Staubli VAL3: Main.pjx

--- Main.pjx ---
Parameters version=s7.8.3 stackSize=10000 millimeterUnit=true
Program file=ContorlLight.pgx
Program file=EnterPageKey.pgx
Program file=Init.pgx
Program file=Main.pgx
Program file=MainKey.pgx
Program file=OnF1.pgx
Program file=OnF2.pgx
Program file=OnF3.pgx
Program file=OnF4.pgx
Program file=OnF5.pgx
Program file=OnF6.pgx
Program file=OnF7.pgx
Program file=OnF8.pgx
Program file=Refresh.pgx
Program file=SetPara.pgx
Program file=start.pgx
Program file=stop.pgx
Data file=Main.dtx
Library alias=user path=Disk://userPage/USERPAGE.pjx
Library alias=RobMaster path=Disk://DealRobMaster/DealRobMaster.pjx
Library alias=Prd path=Disk://Product/Product.pjx
Library alias=Pallet path=Disk://Pallet/Pallet.pjx
Library alias=Path path=Disk://Path/Path.pjx
Library alias=Tool path=Disk://Tool/Tool.pjx autoload=false
Library alias=Frame path=Disk://Frame/Frame.pjx autoload=false
Library alias=IO path=Disk://IO/IO.pjx
Library alias=Home path=Disk://Home/Home.pjx autoload=false
Library alias=PublicData path=Disk://PublicData/PublicData.pjx
Library alias=Motion path=Disk://Motion/Motion.pjx
Library alias=SparePoint path=Disk://SparePoint/SparePoint.pjx autoload=false
Library alias=PublicProg path=Disk://PublicProg/PublicProg.pjx
Library alias=prd path=Disk://template/normalPath/normalPath.pjx

--- Main.dtx ---
mdesc mNomSpeed
bool bExit
bool bUserRefresh
aio aAio
string sParameter
string sListItemValue
bool bListRefresh
string sPath

--- Main.pgx ---
program Main()
  local num l_nKey
begin
  //

  do
    call Refresh()
    l_nKey=getKey()
    bUserRefresh=false
    call MainKey(l_nKey)
    delay(0)
  until bExit
end

--- start.pgx ---
program start()
  local num l_nLastId
  local num l_ni
begin
  call Init()
  taskCreate "light",30,ContorlLight()
  wait(taskStatus("light")==1)
  call Main()
end

--- ContorlLight.pgx ---
program ContorlLight()
begin
  //

  while !bExit
    //红灯
    if PublicData:sStatus=="stop"
      IO:dOut["dOut2"]=true
      IO:dOut["dOut3"]=false
      IO:dOut["dOut4"]=false
    elseIf PublicData:sStatus=="pause"
      IO:dOut["dOut2"]=false
      IO:dOut["dOut3"]=false
      IO:dOut["dOut4"]=true
    elseIf PublicData:sStatus=="run"
      IO:dOut["dOut2"]=false
      IO:dOut["dOut3"]=true
      IO:dOut["dOut4"]=false
    endIf
    delay(0)
  endWhile

end

--- EnterPageKey.pgx ---
program EnterPageKey(num& x_nKey, num& x_nSelect, string& x_sItem)
  local string l_sStr
  local num l_nKey
  local string l_sEmpty
  local string l_sValue
  local num l_nItem
  local num l_nView
  local string l_sItem
  local point lp
  local string l_sYN[2]
  local bool l_bRes
  local num l_nTemp
  local num l_i
begin
  //
  //编辑项目
  switch x_nSelect
    //
    case 0

    break
    //砂带补偿量
    default
      if x_nKey==270
        call user:editNum(x_sItem,sListItemValue[x_nSelect],l_nTemp,x_nSelect)
        if l_nTemp>0.08
          popUpMsg("最大0.08")
          l_nTemp=0.08
          sParameter[x_nSelect]=sPath[x_nSelect-1]
          sListItemValue[0]=toString(".4",PublicData:nDelta)
          call user:strlength(sParameter[l_i],user:nBottomX/2)
          l_sValue=sListItemValue[l_i]
          call user:strlength(l_sValue,user:nBottomX/2+1)
          sParameter[l_i]=sParameter[l_i]+":"+l_sValue
        endIf

        if prd:libLoad("Disk://Traj/"+sPath[x_nSelect-1])==0
          prd:nCompDelta=l_nTemp
          prd:libSave()
        endIf
      endIf

    break
  endSwitch
  if x_nKey==270
    bUserRefresh=true
    bListRefresh=true
  endIf
end

--- Init.pgx ---
program Init()
  local num l_ni
begin
  //
  bExit=false
  bUserRefresh=true
  PublicData:sStatus="stop"
end

--- MainKey.pgx ---
program MainKey(num x_nKey)
  local num l_nKey
begin

  switch x_nKey
    //原始文件转换
    case 271
      call OnF1()
    break
    //路径操作
    case 272
      call OnF2()
    break
    //产品操作
    case 273
      call OnF3()
    break
    //码垛设置
    case 274
      call OnF4()
    break
    //IO
    case 275
      call OnF5()
    break
    //工具/坐标系
    case 276
      call OnF6()
    break
    //生产
    case 277
      call OnF7()
    break
    //退出
    case 278
      call OnF8("是否退出程序")
    break
    //p
    case 112
      call SetPara()
      bUserRefresh=true
    break
  endSwitch
  wait(getKey()==-1)
end

--- OnF1.pgx ---
program OnF1()
begin
  //原始文件
  call RobMaster:start()
  bUserRefresh=true
end

--- OnF2.pgx ---
program OnF2()
begin
  //
  call Path:start()
  bUserRefresh=true
end

--- OnF3.pgx ---
program OnF3()
begin
  call Prd:start()
  bUserRefresh=true
end

--- OnF4.pgx ---
program OnF4()
begin
  call Pallet:start()
  bUserRefresh=true
end

--- OnF5.pgx ---
program OnF5()
begin
  //
  call IO:Main(0)
  bUserRefresh=true
end

--- OnF6.pgx ---
program OnF6()
  local string l_sProperty[4]
  local string l_sItem
begin
  //
  l_sProperty[0]="工具"
  l_sProperty[1]="坐标系"
  l_sProperty[2]="安全点"
  l_sProperty[3]="可用点"
  call user:SetProerty("",26,7,6,4,l_sProperty,l_sItem)
  if l_sItem=="工具"
    Tool:libLoad("Tool")
    call Tool:Main(0)
    Tool:$libClose()
  elseIf l_sItem=="坐标系"
    Frame:libLoad("Frame")
    call Frame:start()
    Frame:$libClose()
  elseIf l_sItem=="安全点"
    Home:libLoad("Home")
    call Home:start()
    Home:$libClose()
  else
    SparePoint:libLoad("SparePoint")
    call SparePoint:start()
    SparePoint:$libClose()
  endIf
  bUserRefresh=true
end

--- OnF7.pgx ---
program OnF7()
begin
  //
  PublicData:bSimulaiton=false
  call Motion:AllMotion(PublicData:sStartPrd)
  PublicData:libSave()
  bUserRefresh=true
end

--- OnF8.pgx ---
program OnF8(string x_sMsg)
  local num l_i
  local string l_sYesNo[2]
begin
  //
  l_sYesNo[0]="是"
  l_sYesNo[1]="否"
  call user:questionDialog(x_sMsg,l_sYesNo,l_i)
  if l_i==0 or l_i==1
    bExit=true
    cls()
  endIf
  bUserRefresh=true
end

--- Refresh.pgx ---
program Refresh()
begin
  //
  if bUserRefresh
    cls()
    userPage()
    gotoxy(1,1)
    put("F1->原始文件转换")
    gotoxy(1,13)
    put("F1")
    gotoxy(1,2)
    put("F2->路径操作")
    gotoxy(6,13)
    put("F2")
    gotoxy(1,3)
    put("F3->产品操作")
    gotoxy(11,13)
    put("F3")
    gotoxy(1,4)
    put("F4->码垛盘设置")
    gotoxy(16,13)
    put("F4")
    gotoxy(1,5)
    put("F5->输入/输出编辑器")
    gotoxy(21,13)
    put("F5")
    gotoxy(1,6)
    put("F6->工具/坐标系/安全点")
    gotoxy(26,13)
    put("F6")
    gotoxy(1,7)
    put("F7->生产")
    gotoxy(31,13)
    put("F7")
    gotoxy(1,8)
    put("F8->退出程序")
    gotoxy(35,13)
    put("F8")

    gotoxy(1,10)
    put("p->参数配置")

  endIf
end

--- SetPara.pgx ---
program SetPara()
  local num l_i
  local num l_nSelect
  local string l_sItem
  local num l_nKey
  local string l_sValue
  local num l_nRes
begin
  //
  cls()
  //获取补偿量列表
  for l_i=0 to size(PublicData:sPrd)-1
    if PublicData:sStartPrd==PublicData:sPrd[l_i]
      call PublicProg:SplitChar(l_nRes,PublicData:sProductList[l_i],"/",sPath)
      l_i=size(PublicData:sPrd)
    endIf
  endFor
  //无匹配产品
  if l_i<size(PublicData:sPrd)+1
    popUpMsg("无启动产品")
    return
  else
    resize(sParameter,1,size(sPath)+1)
    sParameter[0]="产品"
    for l_i=1 to size(sParameter)-1
      sParameter[l_i]=sPath[l_i-1]
    endFor

  endIf

  //
  resize(sListItemValue,1,size(sParameter))
  sListItemValue[0]=PublicData:sStartPrd
  for l_i=1 to size(sParameter)-1
    if prd:libLoad("Disk://Traj/"+sParameter[l_i])==0
      sListItemValue[l_i]=toString(".3",prd:nCompDelta)
    else
      popUpMsg("产品文件"+PublicData:sStartPrd+"错误："+"路径"+sParameter[l_i])
      logMsg("产品文件"+PublicData:sStartPrd+"错误："+"路径"+sParameter[l_i])
      return
    endIf
  endFor

  //
  for l_i=0 to size(sParameter)-1
    call user:strlength(sParameter[l_i],user:nBottomX/2)
    l_sValue=sListItemValue[l_i]
    call user:strlength(l_sValue,user:nBottomX/2+1)
    sParameter[l_i]=sParameter[l_i]+":"+l_sValue
  endFor

  bUserRefresh=true
  bListRefresh=true
  //
  do
    if bUserRefresh
      cls()
      call user:clear(0,13)
      call user:typeMenu(8,"确定")
    endIf
    call user:setList("",sParameter,bUserRefresh,bListRefresh,l_nSelect,l_sItem,l_nKey)
    bListRefresh=bUserRefresh=false
    call EnterPageKey(l_nKey,l_nSelect,sParameter[l_nSelect])
    delay(0)
  until l_nKey==255 or l_nKey==278
  PublicData:libSave()
  bUserRefresh=true
end

--- stop.pgx ---
program stop()
begin
  //
  call IO:CloseAll()
  taskKill("light")
  PublicData:libSave()
end
